{attribute 'GeneratedUsingTerminal: EL1502--0000'}
{attribute addProperty BoxType "EL1502--0000"}
{attribute addProperty Id "EtcSlaveTerminalBaseCNT_InputsAT %I*CNT_Inputs_7D4495CD11CNT_OutputsAT %Q*CNT_Outputs_EB14A6758WcStateAT %I*WcState_9091E0EB2InfoDataAT %I*InfoData_32EB74EA10"}
{attribute addProperty CRC "1054128120"}
{attribute addProperty Size "31"}
TYPE EL1502_3ED4B7F8 EXTENDS EtcSlaveTerminalBase :
STRUCT
	{attribute addProperty Name "CNT_Inputs"}
	CNT_Inputs : CNT_Inputs_7D4495CD;
	{attribute addProperty Name "CNT_Outputs"}
	CNT_Outputs : CNT_Outputs_EB14A675;
	{attribute addProperty Name "WcState"}
	WcState : WcState_9091E0EB;
	{attribute addProperty Name "InfoData"}
	InfoData : InfoData_32EB74EA;
END_STRUCT
END_TYPE

(* stored: Version 1.2.0.0, ProductVersion 3.1.4024.9
   DUT EL1502_3ED4B7F8: Id {d66c17f9-ceee-4f30-be67-12f614b250b4} *)
